(* IEC 61131-3 sources: CODESYS-IO-Visualization/CODESYS-IO-Visualization.fbsproj/Subs/Time, 5 files *)

(* ---- DateTimeStampToString.fn.st ---- *)
FUNCTION DateTimeStampToString : WSTRING

VAR_INPUT
	DateTimeStamp: DateTimeStamp_UDT;
END_VAR

VAR
	tempString: STRING(30);
END_VAR

tempString := CONCAT(TO_STRING(DateTimeStamp.Year),'-');
IF(DateTimeStamp.Month < 10) THEN
	tempString := CONCAT(tempString,'0');
END_IF;
tempString := CONCAT(tempString,TO_STRING(DateTimeStamp.Month));
tempString := CONCAT(tempString,'-');
IF(DateTimeStamp.Day < 10) THEN
	tempString := CONCAT(tempString,'0');
END_IF;
tempString := CONCAT(tempString,TO_STRING(DateTimeStamp.Day));
tempString := CONCAT(tempString,' ');
IF(DateTimeStamp.Hour < 10) THEN
	tempString := CONCAT(tempString,'0');
END_IF;
tempString := CONCAT(tempString,TO_STRING(DateTimeStamp.Hour));
tempString := CONCAT(tempString,':');
IF(DateTimeStamp.Minute < 10) THEN
	tempString := CONCAT(tempString,'0');
END_IF;
tempString := CONCAT(tempString,TO_STRING(DateTimeStamp.Minute));
tempString := CONCAT(tempString,':');
IF(DateTimeStamp.Second < 10) THEN
	tempString := CONCAT(tempString,'0');
END_IF;
tempString := CONCAT(tempString,TO_STRING(DateTimeStamp.Second));

DateTimeStampToString := TO_WSTRING(tempString);

(* ---- PLCClockToString.fn.st ---- *)
FUNCTION PLCClockToString : STRING
VAR_INPUT
	Clock: PLCClock_UDT;
END_VAR
VAR
END_VAR

PLCClockToString := CONCAT(TO_STRING(Clock.Year),'-');
IF(Clock.Month < 10) THEN
	PLCClockToString := CONCAT(PLCClockToString,'0');
END_IF;
PLCClockToString := CONCAT(PLCClockToString,TO_STRING(Clock.Month));
PLCClockToString := CONCAT(PLCClockToString,'-');
IF(Clock.Day < 10) THEN
	PLCClockToString := CONCAT(PLCClockToString,'0');
END_IF;
PLCClockToString := CONCAT(PLCClockToString,TO_STRING(Clock.Day));
PLCClockToString := CONCAT(PLCClockToString,' ');
IF(Clock.Hour < 10) THEN
	PLCClockToString := CONCAT(PLCClockToString,'0');
END_IF;
PLCClockToString := CONCAT(PLCClockToString,TO_STRING(Clock.Hour));
PLCClockToString := CONCAT(PLCClockToString,':');
IF(Clock.Minute < 10) THEN
	PLCClockToString := CONCAT(PLCClockToString,'0');
END_IF;
PLCClockToString := CONCAT(PLCClockToString,TO_STRING(Clock.Minute));
PLCClockToString := CONCAT(PLCClockToString,':');
IF(Clock.Second < 10) THEN
	PLCClockToString := CONCAT(PLCClockToString,'0');
END_IF;
PLCClockToString := CONCAT(PLCClockToString,TO_STRING(Clock.Second));

(* ---- CycleTime.prg.st ---- *)
PROGRAM CycleTime

VAR_IN_OUT
	value: CycleTime_UDT;
END_VAR

value.Now := TIME_TO_DWORD(TIME());

IF (NOT value.init) THEN
	value.init := TRUE;
	value.mSec := 0;
ELSE
	value.mSec := value.Now - value.Last;
END_IF;
value.Last := value.Now;

value.Sec := DWORD_TO_REAL(value.mSec) / 1000.0;

(* ---- GetIsDST.prg.st ---- *)
PROGRAM GetIsDST

VAR_INPUT
	month: INT; (* the current month *)
	day: INT;   (* the current day *)
	hour: INT;  (* the current hour (0 - 23), using Local Standard Time *)
	dow: INT;   (* the day of the week (1 = Monday, 7 = Sunday) using Local Standard Time *)
END_VAR

VAR
	prevSunday: INT;
END_VAR

VAR_OUTPUT
	IsDST: BOOL;
END_VAR

(* DST ON, second Sunday in March, it must be between 3/8 and 3/14 inclusive *)
(* DST OFF, first Sunday in November, it must be between 11/1 and 11/7 inclusive *)

IF (month < 3 OR month > 11) THEN
	IsDST := FALSE;
	RETURN;
END_IF;

IF (month > 3 AND month < 11) THEN
	IsDST := TRUE;
	RETURN;
END_IF;

IF ((month = 11 AND day > 7) OR (month = 3 AND day < 8)) THEN
	IsDST := FALSE;
	RETURN;
END_IF;

IF (month = 3 AND day > 14) THEN
	IsDST := TRUE;
	RETURN;
END_IF;

(* If we get to here, it is either March 8 - 14 or November 1 - 7 *)
prevSunday := day - dow;

IF (month = 3) THEN
	IF (dow = 7) THEN
		IsDST := (hour > 1);
		RETURN;
	END_IF;

	IsDST := (prevSunday > 7 AND prevSunday < 15);
	RETURN;
END_IF;

(* If we get here, it is November 1 - 7 *)
IF (dow = 7) THEN
	IsDST := (hour < 2);
	RETURN;
END_IF;

IsDST := prevSunday < 1;

(* ---- Timer.prg.st ---- *)
PROGRAM Timer

VAR_IN_OUT
	TimerData: Timer_UDT;
END_VAR

VAR
	TimerIn: BOOL;
	TimerPT: TIME;
END_VAR

IF (TimerData.Cancel) THEN
	TimerPT := T#1MS;
	TimerData.Cancel := FALSE;
ELSE
	TimerPT := REAL_TO_TIME(TimerData.PT * 1000.0);
END_IF;

IF (TimerData.Reset) THEN
	TimerIn := FALSE;
	TimerData.Reset := FALSE;
ELSE
	TimerIn := TimerData.In;
END_IF

TimerData.Timer(IN := TimerIn, PT := TimerPT);
TimerData.Q := TimerData.Timer.Q;
TimerData.On := (TimerData.In AND (NOT TimerData.Q));
TimerData.ET := TIME_TO_REAL(TimerData.Timer.ET) / 1000.0;
TimerData.RT := TimerData.PT - TimerData.ET;
